// TwinCAT 3 PLC project Prototype
// ProgramVersion: 3.1.4023.0
// libraries:
//   Tc2_Standard, * (Beckhoff Automation GmbH)
//   Tc2_System, * (Beckhoff Automation GmbH)
//   Tc3_Module, * (Beckhoff Automation GmbH)
// project tree:
//   / Class Diagram_3.TcCD (not stored), PlcTask.TcTTO
//   Classes/ Circle.TcPOU, Rectangle.TcPOU
//   Interfaces/ ITF_Shape.TcIO
//   POUs/ MAIN.TcPOU
// real-time tasks:
//   TASK PlcTask: cycle T#10ms, priority 20, ADS port 350

CONFIGURATION Prototype
    RESOURCE PLC ON TwinCAT3
        TASK PlcTask(INTERVAL := T#10ms, PRIORITY := 20);
        PROGRAM MAIN WITH PlcTask : MAIN;
    END_RESOURCE
END_CONFIGURATION

// ---- Interfaces/ITF_Shape.TcIO
INTERFACE ITF_Shape


METHOD Clone : ITF_Shape
VAR_INPUT
END_VAR
END_METHOD

METHOD Draw
VAR_INPUT
END_VAR
END_METHOD

END_INTERFACE

// ---- POUs/MAIN.TcPOU
PROGRAM MAIN
VAR
    originalRectangle: Rectangle;
    clonedRectangle: ITF_Shape;
	
    originalCircle: Circle;
    clonedCircle: ITF_Shape;
	
	bRequest : BOOL;
	counter: INT;

END_VAR

// https://refactoring.guru/design-patterns/prototype

// Recuerda que el patrón Prototipo permite crear nuevos objetos clonando un objeto existente, evitando así la necesidad de crear nuevas instancias desde cero.

// porque salen varios mensajes:
// https://github.com/tcunit/TcUnit/issues/92
// solución temporal : Unload project...

IF bRequest THEN
	
	originalRectangle.width := 10;
	originalRectangle.height := 5;
	originalRectangle.Draw();
	clonedRectangle := originalRectangle.clone();
	clonedRectangle.Draw();
	
	originalCircle.radius := 7;
	originalCircle.Draw();
	clonedCircle := originalCircle.clone();
	clonedCircle.Draw();
		
	bRequest := FALSE;
//	counter := counter + 1;
//	ADSLOGSTR(msgCtrlMask :=ADSLOG_MSGTYPE_HINT, msgFmtStr :='test: %s', strArg := TO_STRING(counter));
END_IF

END_PROGRAM

// ---- Classes/Rectangle.TcPOU
{attribute 'enable_dynamic_creation'}
FUNCTION_BLOCK Rectangle IMPLEMENTS ITF_Shape
VAR_INPUT
	width: INT;
    height: INT;
END_VAR
VAR_OUTPUT
END_VAR
VAR
END_VAR


METHOD Clone : ITF_Shape
VAR_INPUT
END_VAR
VAR_STAT
	clonedRectangle: Rectangle;
END_VAR
clonedRectangle.width := width;
clonedRectangle.height := height;

Clone := clonedRectangle;
END_METHOD


METHOD Draw

VAR
	str_width : STRING;
	str_height: STRING;
	str : STRING;
END_VAR

str_width  := CONCAT(STR1:= 'width: ', STR2:=  TO_STRING(width));
str_height := CONCAT(STR1:= ', height: ', STR2:=  TO_STRING(height));
str :=  CONCAT(STR1:= str_width, STR2:=  str_height);

ADSLOGSTR(msgCtrlMask :=ADSLOG_MSGTYPE_HINT, msgFmtStr :='Draw Rectangle with:  %s', strArg := str);
END_METHOD

END_FUNCTION_BLOCK

// ---- Classes/Circle.TcPOU
{attribute 'enable_dynamic_creation'}
FUNCTION_BLOCK Circle IMPLEMENTS ITF_Shape
VAR_INPUT
	radius: INT;
END_VAR
VAR_OUTPUT
END_VAR
VAR
END_VAR


METHOD  Clone : ITF_Shape
VAR_INPUT
END_VAR
VAR_STAT
 pClone : POINTER TO Circle;	
END_VAR
pClone := __NEW(Circle);
pClone^.radius := radius;
Clone := pClone^;
__DELETE(pClone);
END_METHOD


METHOD Draw

VAR
	str : STRING;
END_VAR
str := TO_STRING(radius);

ADSLOGSTR(msgCtrlMask :=ADSLOG_MSGTYPE_HINT, msgFmtStr :='Draw circle with radius: %s', strArg := str);
END_METHOD

END_FUNCTION_BLOCK
